{attribute 'hide_all_locals'}
FUNCTION_BLOCK ErrorMover EXTENDS Mover IMPLEMENTS iMover

{attribute 'monitoring' := 'call'}
PROPERTY CurrentDestinationPosition : LREAL
GET


ADSLOGSTR( ADSLOG_MSGTYPE_ERROR, 'The CurrentDestinationPosition Get method has been called on an invalid Mover reference returned by %s.',THIS^.SourceInstancePath);
END_GET
END_PROPERTY

{attribute 'monitoring' := 'call'}
PROPERTY CurrentMoveType : MoverCommandType_enum
GET
VAR
	MoverCurrentMoveType: MoverCommandType_enum;
END_VAR


ADSLOGSTR( ADSLOG_MSGTYPE_ERROR, 'The CurrentMoveType Get method has been called on an invalid Mover reference returned by %s.',THIS^.SourceInstancePath);
END_GET
END_PROPERTY

PROPERTY CurrentObjective : String
GET


ADSLOGSTR( ADSLOG_MSGTYPE_ERROR, 'The CurrentObjective Get method has been called on an invalid Mover reference returned by %s.',THIS^.SourceInstancePath);
END_GET
END_PROPERTY

PROPERTY CurrentTrack : POINTER TO track
GET


ADSLOGSTR( ADSLOG_MSGTYPE_ERROR, 'The CurrentTrack Get method has been called on an invalid Mover reference returned by %s.',THIS^.SourceInstancePath);
END_GET
END_PROPERTY

METHOD Cyclic : iMover
VAR_IN_OUT
	GroupReference		: AXES_GROUP_REF;
END_VAR

VAR
	newCallTime: LREAL;
END_VAR

// If this method was called within the last second, do not write to ADS
newCallTime		:= ULINT_TO_LREAL(F_GetSystemTime())/1E7;

IF ( newCallTime - lastCallCyclic ) > 1 THEN
	ADSLOGSTR( ADSLOG_MSGTYPE_ERROR, 'The Cyclic method has been called on an invalid Mover reference returned by %s.',THIS^.SourceInstancePath);
	lastCallCyclic	:= newCallTime;
END_IF
END_METHOD

METHOD Disable : iMover
VAR_INPUT
END_VAR
VAR
	newCallTime		: LREAL;
END_VAR

// If this method was called within the last second, do not write to ADS
newCallTime		:= ULINT_TO_LREAL(F_GetSystemTime())/1E7;

IF ( newCallTime - lastCallDisable ) > 1 THEN
	ADSLOGSTR( ADSLOG_MSGTYPE_ERROR, 'The Disable method has been called on an invalid Mover reference returned by %s.',THIS^.SourceInstancePath);
	lastCallDisable	:= newCallTime;
END_IF
END_METHOD

METHOD Enable : iMover
VAR_INPUT
END_VAR
VAR
	newCallTime: LREAL;
END_VAR

// If this method was called within the last second, do not write to ADS
newCallTime		:= ULINT_TO_LREAL(F_GetSystemTime())/1E7;

IF ( newCallTime - lastCallEnable ) > 1 THEN
	ADSLOGSTR( ADSLOG_MSGTYPE_ERROR, 'The Enable method has been called on an invalid Mover reference returned by %s.',THIS^.SourceInstancePath);
	lastCallEnable	:= newCallTime;
END_IF
END_METHOD

METHOD GroupStop : iMover
VAR_INPUT
END_VAR
VAR
	newCallTime: LREAL;
END_VAR

// If this method was called within the last second, do not write to ADS
newCallTime		:= ULINT_TO_LREAL(F_GetSystemTime())/1E7;

IF ( newCallTime - lastCallGroupStop ) > 1 THEN
	ADSLOGSTR( ADSLOG_MSGTYPE_ERROR, 'The GroupStop method has been called on an invalid Mover reference returned by %s.',THIS^.SourceInstancePath);
END_IF

lastCallGroupStop	:= newCallTime;
END_METHOD

METHOD Halt : iMover
VAR_INPUT
END_VAR
VAR
	newCallTime: LREAL;
END_VAR

// If this method was called within the last second, do not write to ADS
newCallTime		:= ULINT_TO_LREAL(F_GetSystemTime())/1E7;

IF ( newCallTime - lastCallHalt ) > 1 THEN
	ADSLOGSTR( ADSLOG_MSGTYPE_ERROR, ' The Halt method has been called on an invalid Mover reference returned by %s.',THIS^.SourceInstancePath);
END_IF

lastCallHalt	:= newCallTime;
END_METHOD

{attribute 'monitoring' := 'call'}
PROPERTY IsSyncedToMover : BOOL
GET


ADSLOGSTR( ADSLOG_MSGTYPE_ERROR, 'The IsSyncedToMover Get method has been called on an invalid Mover reference returned by %s.',THIS^.SourceInstancePath);
END_GET
END_PROPERTY

PROPERTY MasterMover : Reference To Mover
GET


ADSLOGSTR( ADSLOG_MSGTYPE_ERROR, 'The MasterMover Get method has been called on an invalid Mover reference returned by %s.',THIS^.SourceInstancePath);
END_GET
END_PROPERTY

METHOD MoveToMultiStation : iMover
VAR_INPUT
	DestinationStation	: REFERENCE TO MultiStation;	
END_VAR
VAR
	newCallTime: LREAL;
END_VAR

// If this method was called within the last second, do not write to ADS
newCallTime		:= ULINT_TO_LREAL(F_GetSystemTime())/1E7;

IF ( newCallTime - lastCallMovePos ) > 1 THEN
	ADSLOGSTR( ADSLOG_MSGTYPE_ERROR, 'The MoveToStation method has been called on an invalid Mover reference returned by %s.',THIS^.SourceInstancePath);
	lastCallMovePos		:= newCallTime;
END_IF
END_METHOD

METHOD PUBLIC MoveToPosition : iMover
VAR_INPUT
	DestinationPosition		: LREAL;	// position on track for a shuttle to move towards
END_VAR
VAR
	newCallTime				: LREAL;
END_VAR

// If this method was called within the last second, do not write to ADS
newCallTime		:= ULINT_TO_LREAL(F_GetSystemTime())/1E7;

IF ( newCallTime - lastCallMovePos ) > 1 THEN
	ADSLOGSTR( ADSLOG_MSGTYPE_ERROR, 'The MoveToPosition method has been called on an invalid Mover reference returned by %s.',THIS^.SourceInstancePath);
	lastCallMovePos		:= newCallTime;
END_IF
END_METHOD

METHOD MoveToStation : iMover
VAR_INPUT
	DestinationStation	: REFERENCE TO Station;	
END_VAR
VAR
	newCallTime: LREAL;
END_VAR

// If this method was called within the last second, do not write to ADS
newCallTime		:= ULINT_TO_LREAL(F_GetSystemTime())/1E7;

IF ( newCallTime - lastCallMovePos ) > 1 THEN
	ADSLOGSTR( ADSLOG_MSGTYPE_ERROR, 'The MoveToStation method has been called on an invalid Mover reference returned by %s.',THIS^.SourceInstancePath);
	lastCallMovePos		:= newCallTime;
END_IF
END_METHOD

METHOD MoveVelocity : iMover
VAR_INPUT
	DesiredVelocity : LREAL;		//The velocity to be commanded [mm/s]
END_VAR

VAR
	negativeCommand: BOOL;
	newCallTime: LREAL;
END_VAR

// If this method was called within the last second, do not write to ADS
newCallTime		:= ULINT_TO_LREAL(F_GetSystemTime())/1E7;

IF ( newCallTime - lastCallMoveVel ) > 1 THEN
	ADSLOGSTR( ADSLOG_MSGTYPE_ERROR, 'The MoveVelocity method has been called on an invalid Mover reference returned by %s.',THIS^.SourceInstancePath);
	lastCallMoveVel		:= newCallTime;
END_IF
END_METHOD

PROPERTY Payload : USINT
GET


ADSLOGSTR( ADSLOG_MSGTYPE_ERROR, 'The Payload Get method has been called on an invalid Mover reference returned by %s.',THIS^.SourceInstancePath);
END_GET
SET


ADSLOGSTR( ADSLOG_MSGTYPE_ERROR, 'The Payload Set method has been called on an invalid Mover reference returned by %s.',THIS^.SourceInstancePath);
END_SET
END_PROPERTY

METHOD ReissueCommand : iMover
VAR_INPUT
END_VAR

VAR
	newCallTime: LREAL;
END_VAR

// If this method was called within the last second, do not write to ADS
newCallTime		:= ULINT_TO_LREAL(F_GetSystemTime())/1E7;

IF ( newCallTime - lastCallReissue ) > 1 THEN
	ADSLOGSTR( ADSLOG_MSGTYPE_ERROR, 'The ReissueCommand method has been called on an invalid Mover reference returned by %s.',THIS^.SourceInstancePath);
	lastCallReissue		:= newCallTime;
END_IF
END_METHOD

METHOD SetAcceleration : iMover
VAR_INPUT
	Acceleration	: LREAL;
END_VAR

VAR
	newCallTime: LREAL;
END_VAR

// If this method was called within the last second, do not write to ADS
newCallTime		:= ULINT_TO_LREAL(F_GetSystemTime())/1E7;

IF ( newCallTime - lastCallSetAcc ) > 1 THEN
	ADSLOGSTR( ADSLOG_MSGTYPE_ERROR, 'The SetAcceleration method has been called on an invalid Mover reference returned by %s.',THIS^.SourceInstancePath);
	lastCallSetAcc		:= newCallTime;
END_IF
END_METHOD

METHOD SetDeceleration : iMover
VAR_INPUT
	Deceleration	: LREAL;
END_VAR

VAR
	newCallTime: LREAL;
END_VAR

// If this method was called within the last second, do not write to ADS
newCallTime		:= ULINT_TO_LREAL(F_GetSystemTime())/1E7;

IF ( newCallTime - lastCallSetDec ) > 1 THEN
	ADSLOGSTR( ADSLOG_MSGTYPE_ERROR, 'The SetDeceleration method has been called on an invalid Mover reference returned by %s.',THIS^.SourceInstancePath);
	lastCallSetDec		:= newCallTime;
END_IF
END_METHOD

METHOD SetDirection : iMover
VAR_INPUT
	Direction		: Tc3_Mc3Definitions.MC_Direction;
END_VAR

VAR
	newCallTime: LREAL;
END_VAR

// If this method was called within the last second, do not write to ADS
newCallTime		:= ULINT_TO_LREAL(F_GetSystemTime())/1E7;

IF ( newCallTime - lastCallSetDir ) > 1 THEN
	ADSLOGSTR( ADSLOG_MSGTYPE_ERROR, 'The SetDirection method has been called on an invalid Mover reference returned by %s.',THIS^.SourceInstancePath);
	lastCallSetDir		:= newCallTime;
END_IF
END_METHOD

METHOD SetJerk : iMover
VAR_INPUT
	Jerk		: LREAL;
END_VAR

VAR
	newCallTime: LREAL;
END_VAR

// If this method was called within the last second, do not write to ADS
newCallTime		:= ULINT_TO_LREAL(F_GetSystemTime())/1E7;

IF ( newCallTime - lastCallSetJerk ) > 1 THEN
	ADSLOGSTR( ADSLOG_MSGTYPE_ERROR, 'The SetJerk method has been called on an invalid Mover reference returned by %s.',THIS^.SourceInstancePath);
	lastCallSetJerk		:= newCallTime;
END_IF
END_METHOD

METHOD SetVelocity : iMover
VAR_INPUT
	Velocity	: LREAL;
END_VAR

VAR
	newCallTime: LREAL;
END_VAR

// If this method was called in the last second, do not write to ADS
newCallTime		:= ULINT_TO_LREAL(F_GetSystemTime())/1E7;

IF ( newCallTime - lastCallSetVel ) > 1 THEN
	ADSLOGSTR( ADSLOG_MSGTYPE_ERROR, 'The SetVelocity method has been called on an invalid Mover reference returned by %s.',THIS^.SourceInstancePath);
	lastCallSetVel		:= newCallTime;
END_IF
END_METHOD

METHOD SyncToAxis : iMover
VAR_INPUT
	
	MasterAxis		: REFERENCE TO AXIS_REF;
	MasterSyncPos	: LREAL;	// Master sync position (nonmodulo), where the input axis will be located when first synchronized
	SlaveSyncPos	: LREAL;	// Mover sync position, where the mover will be located when first synchronized
	SyncStrategy	: MC_SYNC_STRATEGY;	// Direction input
	
END_VAR
VAR
	newCallTime		: LREAL;
END_VAR


// If this method was called within the last second, do not write to ADS
newCallTime		:= ULINT_TO_LREAL(F_GetSystemTime())/1E7;

IF (newCallTime - lastCallSync) > 1 THEN
	ADSLOGSTR( ADSLOG_MSGTYPE_ERROR,'The SyncToAxis method has been called on an invalid Mover reference returned by %s',THIS^.SourceInstancePath);
	lastCallSync		:= newCallTime;
END_IF
END_METHOD

METHOD SyncToMover : iMover
VAR_INPUT

	MasterMover		: REFERENCE TO Mover;	// Synchronization master mover, whose position to follow. Further motion commands break the pairing
	Gap				: LREAL;				// Gap distance to lead mover. Positive values indicate following, negative values indicate leading

END_VAR

VAR
	newCallTime: LREAL;
END_VAR

// IF this method was called within the last second, do not write to ADS
newCallTime		:= ULINT_TO_LREAL(F_GetSystemTime())/1E7;

IF ( newCallTime - lastCallSync ) > 1 THEN
	ADSLOGSTR( ADSLOG_MSGTYPE_ERROR, 'The SyncToMover method has been called on an invalid Mover reference returned by %s.',THIS^.SourceInstancePath);
	lastCallSync	:= newCallTime;
END_IF
END_METHOD

END_FUNCTION_BLOCK

(* stored: Version 1.1.0.1, ProductVersion 3.1.4024.12
   POU ErrorMover: Id {bd3df610-8473-440e-a9dc-a09f811846e0}, SpecialFunc None
   Folder Methods: Id {95344208-9410-4fde-9b34-506fa304a287}
   Folder Properties: Id {6fd2fbdb-965d-489f-acb7-82704f375aa0}
   Property CurrentDestinationPosition: Id {2b4b67cc-3100-4b95-930e-6d7f88a409da}
   Get Get: Id {4ab8604e-f7e5-4051-87ad-121e3916f22d}
   Property CurrentMoveType: Id {654cf008-4e25-44e0-a02e-14f98c95c229}
   Get Get: Id {ff80f46a-8539-4feb-9642-1a61fe0c4d1f}
   Property CurrentObjective: Id {7897b829-22ce-468b-bc00-104f4387a246}
   Get Get: Id {43ffd29e-7106-4bdc-961e-f77ce36447cf}
   Property CurrentTrack: Id {9bc4654e-1097-0e57-303b-26deb5d985c1}
   Get Get: Id {00e132d6-ae6d-07ef-39af-0aace549cb59}
   Method Cyclic: Id {764e6bb0-4d0d-42b1-82a2-beacd8ec9b5d}
   Method Disable: Id {a35f8faa-093e-4292-a444-f58b6f5f6d4f}
   Method Enable: Id {d4744d94-4a3b-451e-bbfc-59a59ee494e3}
   Method GroupStop: Id {4e389025-4e76-4cce-ac5c-8a82b786913e}
   Method Halt: Id {8cf1fd35-c92c-43a7-89e5-e709149394be}
   Property IsSyncedToMover: Id {6b623c29-8901-4623-afb3-f30839740c89}
   Get Get: Id {11e533df-3e35-43ba-a245-0cb48a9f5be4}
   Property MasterMover: Id {6243eebd-fe41-4008-9c02-b6d5bac54829}
   Get Get: Id {763be082-226a-441a-8e70-1d4aacb4d1ea}
   Method MoveToMultiStation: Id {09d9ee59-8c45-0f46-0ef9-6c67164988f7}
   Method MoveToPosition: Id {06584b48-b7d7-45ec-b670-d5553ed7efde}
   Method MoveToStation: Id {f7d51585-b63e-4a40-86ce-600a20ecf081}
   Method MoveVelocity: Id {6f39fd6e-0630-4b12-9284-3c4d7e063735}
   Property Payload: Id {24ebdcd3-9649-41f7-9f65-e4f7f86ef316}
   Get Get: Id {28f7f04b-9925-4df5-91ef-030257222faa}
   Set Set: Id {0f0e05f2-3b7b-4da0-bed5-5c8e12c1a732}
   Method ReissueCommand: Id {2b2633c0-7db7-4352-ae48-063856e2b0db}
   Method SetAcceleration: Id {90f501cd-2aae-43a2-a87f-fdbe1a4cb2d2}
   Method SetDeceleration: Id {1da65927-f09e-4d2d-9427-dff6efde0728}
   Method SetDirection: Id {2ad42cfb-45f4-4a68-956c-6004efe4ef84}
   Method SetJerk: Id {8f7db2a4-6343-4dd3-aa2a-28dea1975f9e}
   Method SetVelocity: Id {cdd1b3bc-a3c7-4bf5-8a9b-c45db8a075f7}
   Method SyncToAxis: Id {cfaf0d71-8323-03cc-05f8-4e7eec7d0bc9}
   Method SyncToMover: Id {cd1d5b64-e134-455b-8660-842288b989a0} *)
